INTERFACE I_DatatypeOperation EXTENDS I_Disposable

METHOD Execute
VAR
END_VAR
END_METHOD

END_INTERFACE

(* stored: Version 1.1.0.1, ProductVersion 3.1.4024.12
   Itf I_DatatypeOperation: Id {e5f08455-1773-465e-9fdd-0194beaa9a1e}
   Method Execute: Id {24fd2133-75ab-44e2-a2b8-a4bd04ec95fd} *)
